SYSTEM TEST_SYSTEM (* Test adding FB to Device *)
  (* Standard: 61499-1 *)
  (* Version 0.0, 2006-03-22, JHC, Holobloc Inc, Test adding FB to Device. *)
  APPLICATION APP1
  END_APPLICATION
  DEVICE DEV1 : DeviceType
    RESOURCE RES2 : ResourceType
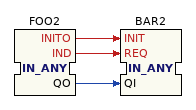
      FBS
        FOO2 : IN_ANY;
        BAR2 : IN_ANY;
      END_FBS
      EVENT_CONNECTIONS
        FOO2.INITO TO BAR2.INIT;
        FOO2.IND TO BAR2.REQ;
      END_CONNECTIONS
      DATA_CONNECTIONS
        FOO2.QO TO BAR2.QI;
      END_CONNECTIONS
    END_RESOURCE
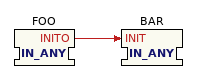
    [picture p1: device DEV1]
    FBS
      FOO : IN_ANY;
      BAR : IN_ANY;
    END_FBS
    EVENT_CONNECTIONS
      FOO.INITO TO BAR.INIT;
    END_CONNECTIONS
  END_DEVICE
END_SYSTEM
